// SIMATIC S7-200 project (STEP 7-Micro/WIN), CPU 224XP REL 02.01

SYMBOL_TABLE 用户定义1
控制模式             VW0      //
设定值              VD100
反馈               VD104
手动值              VD108
P参数              VD112
I参数              VD116
D参数              VD120
显示输的百分比          VD124
输出值              VW200
END_SYMBOL_TABLE

ORGANIZATION_BLOCK 主程序:OB1
TITLE=程序注释
BEGIN
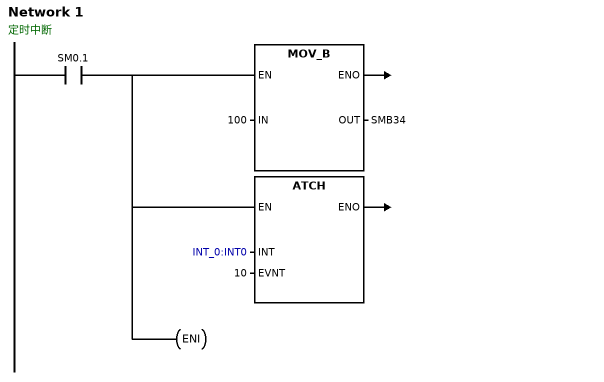
Network 1
// 定时中断
LD     SM0.1
MOVB   100, SMB34
ATCH   INT_0:INT0, 10
ENI
Network 2 // 网络标题
// 网络注释
END_ORGANIZATION_BLOCK

SUBROUTINE_BLOCK PID_1:SBR9
TITLE=
VAR_INPUT
con_mofe:WORD;	// LW0   控制模式
theset:REAL;	// LD2   设置
feedback:REAL;	// LD6   反馈
hand_set:REAL;	// LD10   手动设置
P:REAL;	// LD14 P参数
I:REAL;	// LD18 I参数
D:REAL;	// LD22 D参数
END_VAR
VAR_OUTPUT
out_val:REAL;	// LD26   输出_显示
out_int:INT;	// LW30   输出_AQW
END_VAR
VAR
thewarp:REAL;	// LD32   当前误差
twowarp:REAL;	// LD36   两次偏差
I_out:REAL;	// LD40 
D_out:REAL;	// LD44 
P_out:REAL;	// LD48 
TEMP1:DINT;	// LD52 
END_VAR
BEGIN
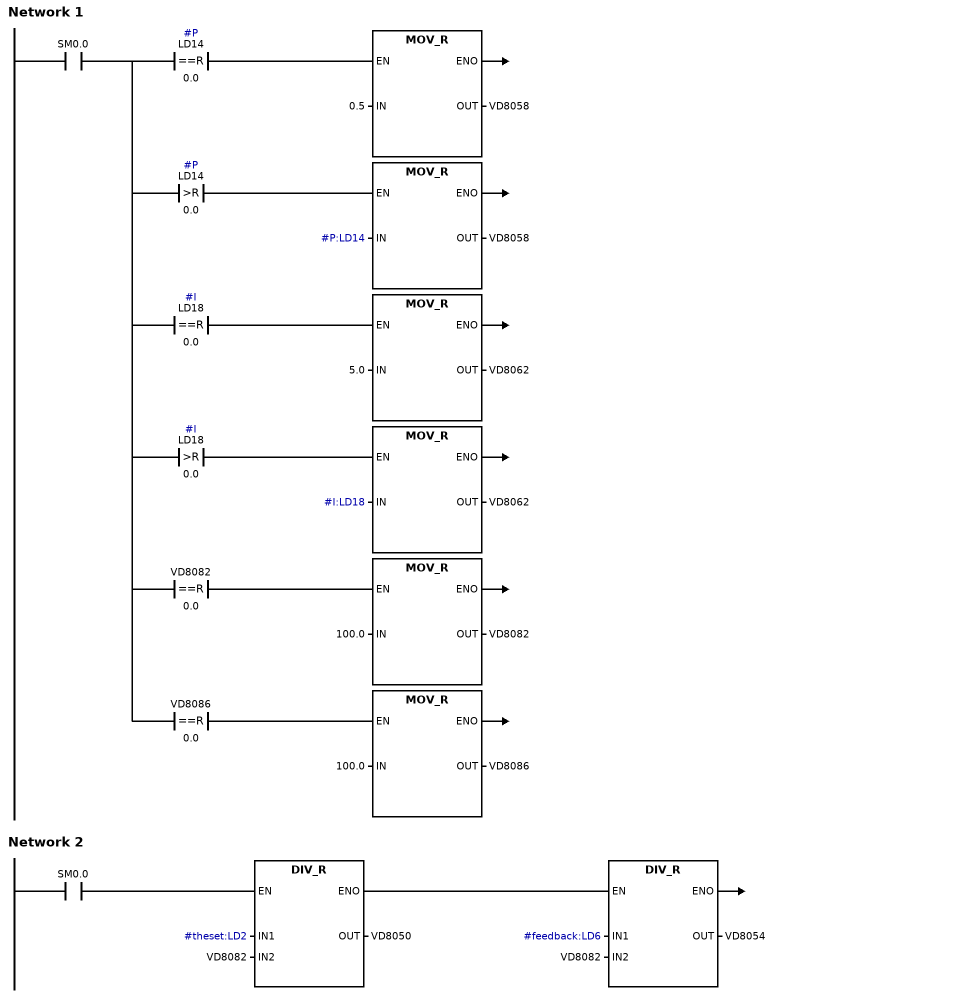
Network 1
LD     SM0.0
LPS
AR=    #P:LD14, 0.0
MOVR   0.5, VD8058
LRD
AR>    #P:LD14, 0.0
MOVR   #P:LD14, VD8058
LRD
AR=    #I:LD18, 0.0
MOVR   5.0, VD8062
LRD
AR>    #I:LD18, 0.0
MOVR   #I:LD18, VD8062
LRD
AR=    VD8082, 0.0
MOVR   100.0, VD8082
LPP
AR=    VD8086, 0.0
MOVR   100.0, VD8086
Network 2
LD     SM0.0
MOVR   #theset:LD2, VD8050
AENO
/R     VD8082, VD8050
AENO
MOVR   #feedback:LD6, VD8054
/R     VD8082, VD8054
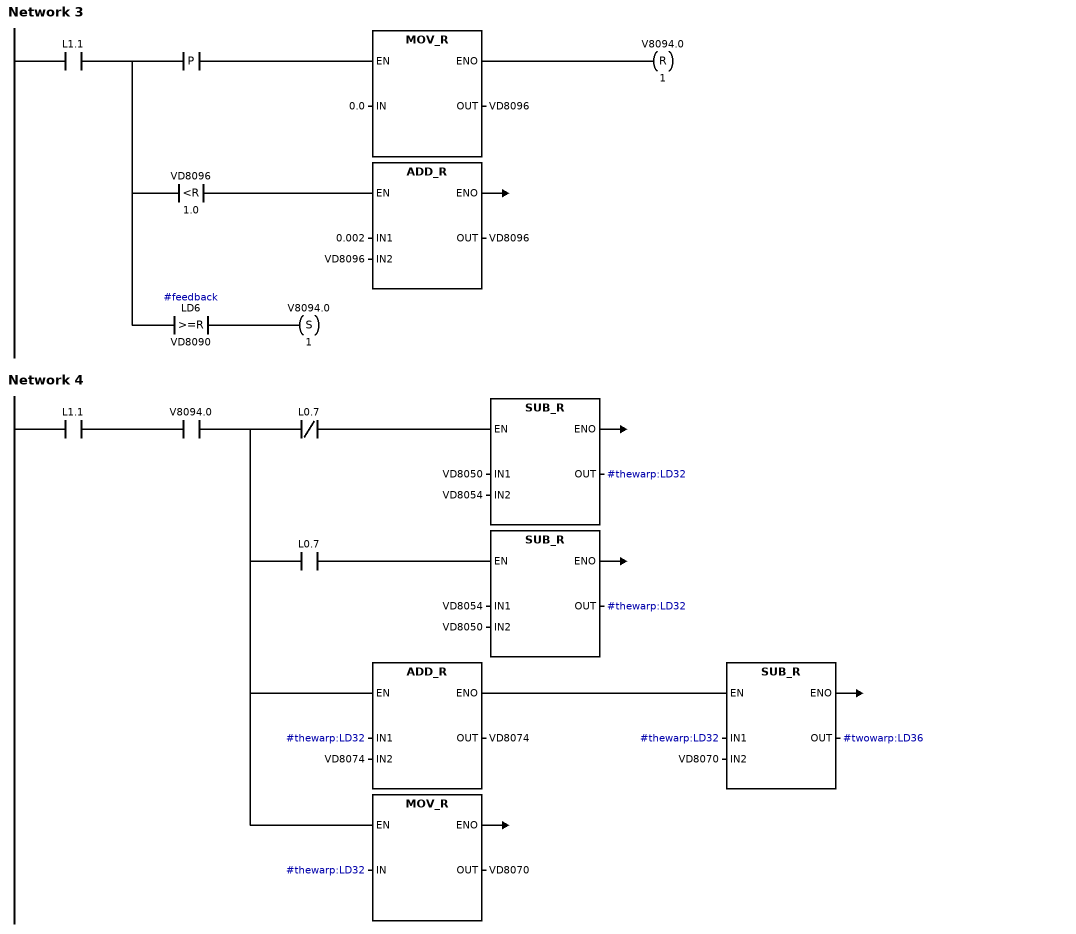
Network 3
LD     L1.1
LPS
EU
MOVR   0.0, VD8096
AENO
R      V8094.0, 1
LRD
AR<    VD8096, 1.0
+R     0.002, VD8096
LPP
AR>=   #feedback:LD6, VD8090
S      V8094.0, 1
Network 4
LD     L1.1
A      V8094.0
LPS
AN     L0.7
MOVR   VD8050, #thewarp:LD32
-R     VD8054, #thewarp:LD32
LRD
A      L0.7
MOVR   VD8054, #thewarp:LD32
-R     VD8050, #thewarp:LD32
LRD
+R     #thewarp:LD32, VD8074
AENO
MOVR   #thewarp:LD32, #twowarp:LD36
-R     VD8070, #twowarp:LD36
LPP
MOVR   #thewarp:LD32, VD8070
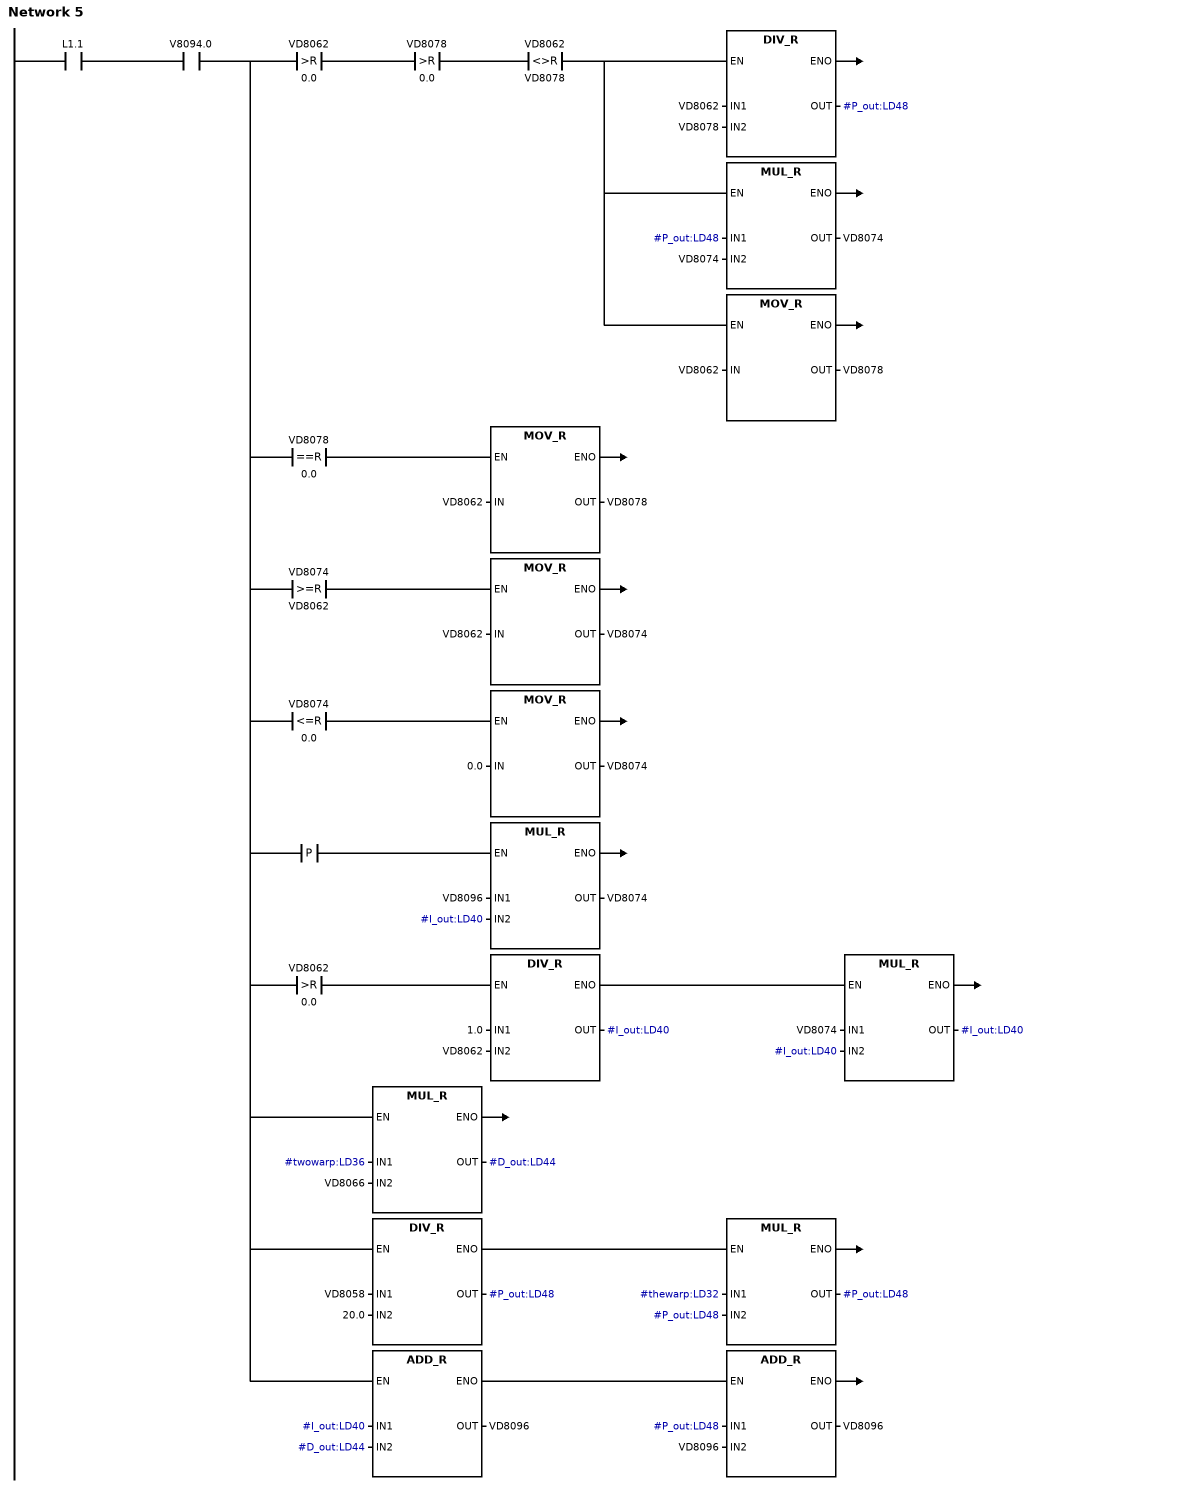
Network 5
LD     L1.1
A      V8094.0
LPS
AR>    VD8062, 0.0
AR>    VD8078, 0.0
AR<>   VD8062, VD8078
MOVR   VD8062, #P_out:LD48
/R     VD8078, #P_out:LD48
*R     #P_out:LD48, VD8074
MOVR   VD8062, VD8078
LPP
LPS
AR=    VD8078, 0.0
MOVR   VD8062, VD8078
LRD
AR>=   VD8074, VD8062
MOVR   VD8062, VD8074
LRD
AR<=   VD8074, 0.0
MOVR   0.0, VD8074
LRD
EU
MOVR   VD8096, VD8074
*R     #I_out:LD40, VD8074
LRD
AR>    VD8062, 0.0
MOVR   1.0, #I_out:LD40
AENO
/R     VD8062, #I_out:LD40
AENO
*R     VD8074, #I_out:LD40
LRD
MOVR   #twowarp:LD36, #D_out:LD44
*R     VD8066, #D_out:LD44
LRD
MOVR   VD8058, #P_out:LD48
AENO
/R     20.0, #P_out:LD48
AENO
*R     #thewarp:LD32, #P_out:LD48
LPP
MOVR   #I_out:LD40, VD8096
AENO
+R     #D_out:LD44, VD8096
AENO
+R     #P_out:LD48, VD8096
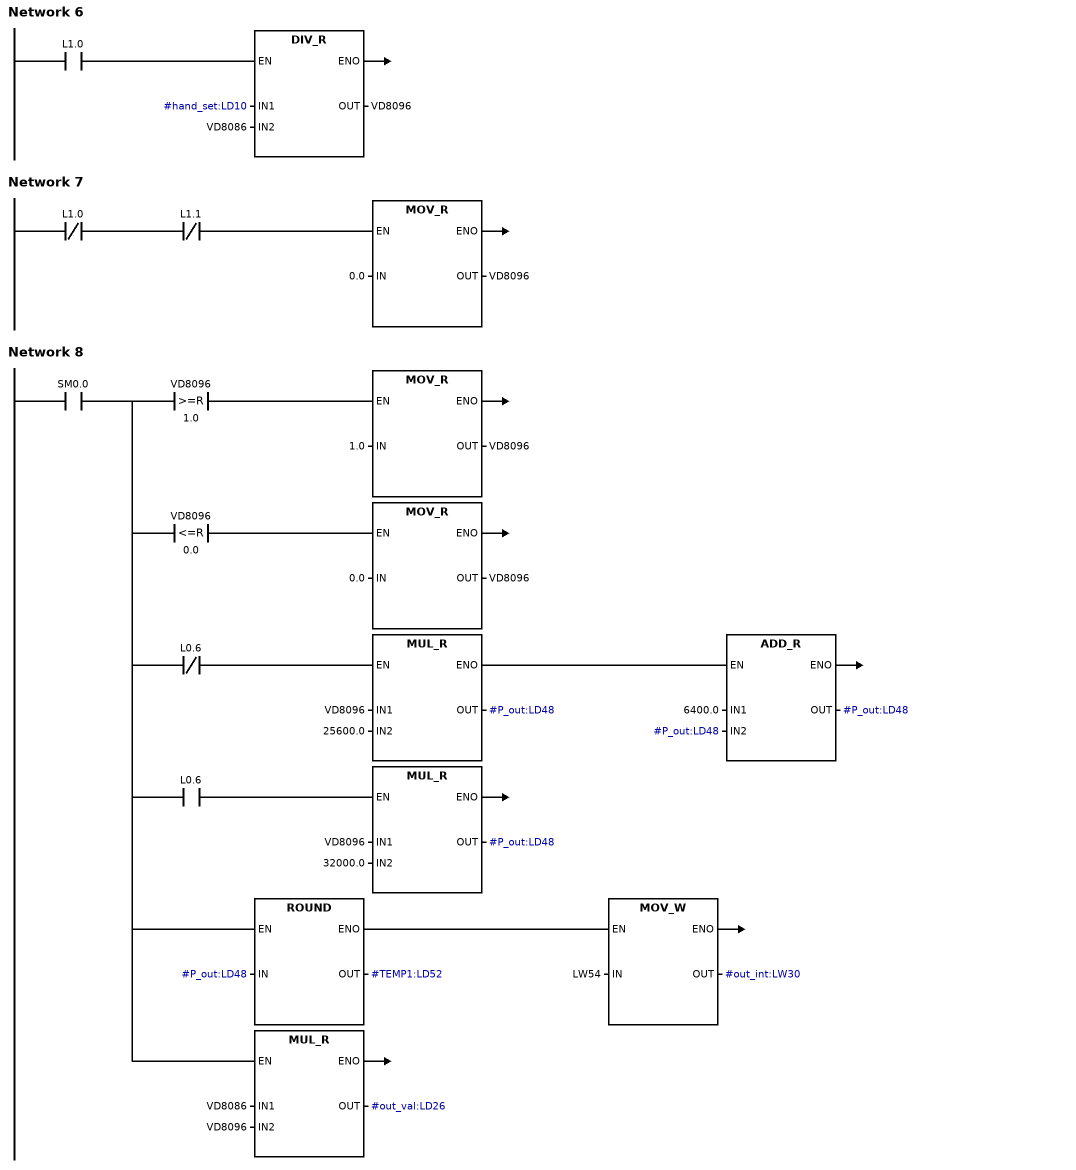
Network 6
LD     L1.0
MOVR   #hand_set:LD10, VD8096
/R     VD8086, VD8096
Network 7
LDN    L1.0
AN     L1.1
MOVR   0.0, VD8096
Network 8
LD     SM0.0
LPS
AR>=   VD8096, 1.0
MOVR   1.0, VD8096
LRD
AR<=   VD8096, 0.0
MOVR   0.0, VD8096
LRD
AN     L0.6
MOVR   VD8096, #P_out:LD48
AENO
*R     25600.0, #P_out:LD48
AENO
+R     6400.0, #P_out:LD48
LRD
A      L0.6
MOVR   VD8096, #P_out:LD48
*R     32000.0, #P_out:LD48
LRD
ROUND  #P_out:LD48, #TEMP1:LD52
AENO
MOVW   LW54, #out_int:LW30
LPP
MOVR   VD8086, #out_val:LD26
*R     VD8096, #out_val:LD26
END_SUBROUTINE_BLOCK

INTERRUPT_BLOCK INT_0:INT0
TITLE=中断程序注释
BEGIN
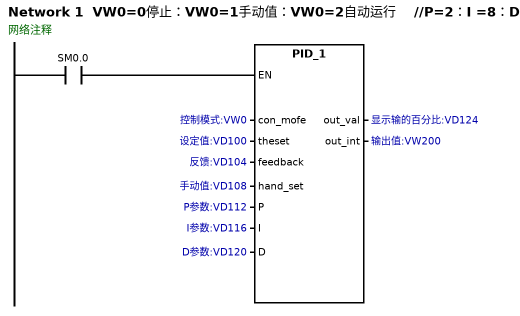
Network 1 // VW0=0停止：VW0=1手动值：VW0=2自动运行    //P=2：I =8：D=0
// 网络注释
LD     SM0.0
CALL   PID_1:SBR9, 控制模式:VW0, 设定值:VD100, 反馈:VD104, 手动值:VD108, P参数:VD112, I参数:VD116, D参数:VD120, 显示输的百分比:VD124, 输出值:VW200
END_INTERRUPT_BLOCK
